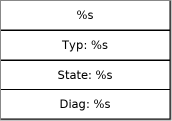
VISUALIZATION TplTsFb  // 172x121
VAR_IN_OUT
	stfbDiag 					:FB_TwinSafeFB;
END_VAR
(* End *)
    Rectangle (0,0 170x30), "%s", text variable: stfbDiag.sName, colour toggle: stfbDiag.sState = 'RUN' or stfbDiag.sState = 'MON_ON'
    Rectangle (0,30 170x30), "Typ: %s", text variable: stfbDiag.sType
    Rectangle (0,60 170x30), "State: %s", text variable: stfbDiag.sState, colour toggle: stfbDiag.sState = 'ERROR'
    Rectangle (0,89 170x30), "Diag: %s", text variable: stfbDiag.sDiag
END_VISUALIZATION

(* stored: Version 1.1.0.1, ProductVersion 3.1.4024.11
   Visu TplTsFb: Id {1bf462fc-40bd-4812-a7fd-7eafc8b12c37} *)
